FUNCTION_BLOCK Test_TStreamAdd_Read_PVOID_CheckAlignment EXTENDS T_UnitTestBase
VAR
    Stream  : T_Stream(StreamLength := 2);
    ArgType : E_ArgTypeId := E_ArgTypeId.Type_PVOID;
    Bob     : INT;
END_VAR

{attribute 'analysis' := '-33'} // inhibit unused variable warning
METHOD RunTest
IF Retest THEN
    SUPER^.Init();
END_IF

IF TestCompleted THEN
    RETURN;
END_IF

F_Inc(CycleCount);
IF CycleCount > 1000 THEN
    Fail(Message := 'Timeout');
END_IF

Stream.Init(2);

Stream.Add_BYTE(123);// add a byte to test alignment checks...
Stream.Add_PVOID(ADR(Bob));

Stream.SetReadPosition(0);

Stream.Read_BYTE();

// check next value...	
AssertEquals_PVOID(Expected     := ADR(Bob),
                             Actual       := Stream.Read_PVOID(),
                             Message := 'Stream.Read_PVOID()');

// check we are at the end of the stream..							
AssertEquals_UDINT(Expected     := Stream.StreamLength,
                             Actual       := Stream.ReadPosition,
                             Message := 'Stream.ReadPosition');

TestCompleted := TRUE;
END_METHOD

END_FUNCTION_BLOCK

(* stored: Version 1.1.0.1, ProductVersion 3.1.4024.15
   POU Test_TStreamAdd_Read_PVOID_CheckAlignment: Id {acf46996-4dfc-4d27-ad64-59556ad8f864}, SpecialFunc None
   Method RunTest: Id {91e66146-7b52-4f15-9c69-8591d1ade112} *)
